{attribute 'qualified_only'}
{attribute 'strict'}
TYPE MOTION_STATE :
(
	JOGGING_UP,
	JOGGING_DOWN,
	AUTO,
	MOVE_COMPLETE
);
END_TYPE

(* stored: Version 1.1.0.1, ProductVersion 3.1.4022.12
   DUT MOTION_STATE: Id {151b387b-7321-4206-918a-c6840c3ef8fa} *)
